(* PLC project product, Dassault Systèmes ControlBuild 2024x *)
(* stored: creationDateTime 2023-10-04T11:03:57-01:00 *)

(* This module simulates a generic product "box". *)
FUNCTION_BLOCK motion_control.product
  VAR
    status_act_prod : DINT := 0;
    m11 : REAL := 1.0;
    m12 : REAL := 0.0;
    m13 : REAL := 0.0;
    m14 : REAL := 0.0;
    m21 : REAL := 0.0;
    m22 : REAL := 1.0;
    m23 : REAL := 0.0;
    m24 : REAL := 0.0;
    m31 : REAL := 0.0;
    m32 : REAL := 0.0;
    m33 : REAL := 1.0;
    m34 : REAL := 0.0;
    m41 : REAL := 0.0;
    m42 : REAL := 0.0;
    m43 : REAL := 0.0;
    m44 : REAL := 1.0;
    movementConv : REAL := 0.0;
    contact : BOOL := false;
    centreRotX : REAL := 0.0;
    centreRotZ : REAL := 0.0;
    centreRotY : REAL := 0.0;
    moveDirection : INT := 0;
    idConv : DINT := 0;
    moveAuthorization : BOOL := false;
    number : INT := 0;
    idProdBelow : DINT := 0;
    prodId : INT := 0;
    oldOtherPx : REAL := 0.0;
    oldOtherPy : REAL := 0.0;
    oldOtherPz : REAL := 0.0;
    oldOtherRx : REAL := 0.0;
    oldOtherRy : REAL := 0.0;
    oldOtherRz : REAL := 0.0;
    gravitySpeed : REAL := 0.0;
    oldIdConv : DINT := 0;
  END_VAR
  VAR
    display1 : INT := 0;
    display2 : INT := 0;
    display3 : INT := 0;
    display4 : INT := 0;
    display5 : INT := 0;
    display6 : INT := 0;
    display7 : INT := 0;
    display8 : INT := 0;
    display9 : INT := 0;
    display10 : INT := 0;
  END_VAR
  VAR
    oPx : REAL := 0.0;
    oPy : REAL := 0.0;
    oPz : REAL := 0.0;
    oAx : REAL := 0.0;
    oAy : REAL := 0.0;
    oAz : REAL := 0.0;
    armActive : BOOL := false;
    memArmActive : BOOL := false;
    refAngZ : REAL := 0.0;
    refAngY : REAL := 0.0;
    refAngX : REAL := 0.0;
    refZ : REAL := 0.0;
    refY : REAL := 0.0;
    refX : REAL := 0.0;
    refSizeOthX : REAL := 0.0;
    refAngOthZ : REAL := 0.0;
    refAngOthY : REAL := 0.0;
    refAngOthX : REAL := 0.0;
    refOthZ : REAL := 0.0;
    refOthY : REAL := 0.0;
    refOthX : REAL := 0.0;
  END_VAR
  VAR
    empty1 : BOOL := false;
    empty2 : BOOL := false;
    empty3 : BOOL := false;
    empty4 : BOOL := false;
    empty5 : BOOL := false;
    empty6 : BOOL := false;
    empty7 : BOOL := false;
    empty8 : BOOL := false;
  END_VAR
  VAR
    weight : INT := 0;
  END_VAR


ACTION Prelude:
/* ----------------------------------------------------------------	*/
/* Initialisation of local variables of the instance of the product	*/
/* ----------------------------------------------------------------	*/
weight =0;
movementConv = 0.0;
contact = 0;
moveAuthorization = 1;
idConv=-1;
armActive = 0;

if (!empty1) weight +=15;
if (!empty2) weight +=15;
if (!empty3) weight +=15;
if (!empty4) weight +=15;
if (!empty5) weight +=15;
if (!empty6) weight +=15;
if (!empty7) weight +=15;
if (!empty8) weight +=15;
END_ACTION

ACTION Postlude:
/* ----------------------------------------------------------------	*/
/* If there is no contact, the box falls down thanks to gravity	*/	
/* ----------------------------------------------------------------	*/
if (contact == 0) 
	moveZBy(myself, gravitySpeed*-1.0);


/* ----------------------------------------------------------------	*/
/* Shift on conveyors if authorization					*/
/* ----------------------------------------------------------------	*/
if (moveAuthorization == 1 && (idConv>=0)) 
	moveRelativeAnotherBy(myself, idConv, movementConv, 0.0, 0.0);


/* ----------------------------------------------------------------	*/
/* Reset memories								*/
/* ----------------------------------------------------------------	*/
if (contact == 0) {
	moveDirection = 0;
	idProdBelow = -1;
}

memArmActive = armActive;
END_ACTION

ACTION motion_lib.qrreader:
otherVar(number) = number;
END_ACTION

ACTION motion_lib.weighingscale:
otherVar(weight) = weight;
END_ACTION

ACTION motion_lib.pusher:
moveBy(myself , otherVar(moveX1),otherVar(moveY1) , otherVar(moveZ1));
END_ACTION

ACTION motion_control.robotic_arm:
armActive = otherVar(functionActiveLocale);
if (armActive && !memArmActive ) {

// --- take arm/product relative position reference ---
	refOthX = getPositionX(other);
	refOthY = getPositionY(other);
	refOthZ = getPositionZ(other);
	refAngOthX = getAngleX(other);
	refAngOthY = getAngleY(other);
	refAngOthZ = getAngleZ(other);
	refSizeOthX = getSizeX(other);
	
	// move myself to the arm space reference 
	moveBy(myself, -refOthX, -refOthY, -refOthZ);

	rotateZBy(myself,-refAngOthZ,0.0, 0.0, 0.0);
	rotateYBy(myself,-refAngOthY,0.0, 0.0, 0.0);
	rotateXBy(myself,-refAngOthX,0.0, 0.0, 0.0);

	refX = getPositionX(myself);
	refY = getPositionY(myself);
	refZ = getPositionZ(myself);
	refAngX = getAngleX(myself);
	refAngY = getAngleY(myself);
	refAngZ = getAngleZ(myself);

	rotateBy(myself,refAngOthX,refAngOthY, refAngOthZ, 0.0, 0.0, 0.0); // relocate the product
	moveBy(myself, refOthX, refOthY, refOthZ);
}

if (armActive && memArmActive) {
	rotateTo(myself,refAngX,refAngY,refAngZ, getPositionX(myself), getPositionY(myself), getPositionZ(myself));
	moveTo(myself, refX, refY, refZ);
	rotateBy(myself,getAngleX(other),getAngleY(other), getAngleZ(other), 0.0, 0.0, 0.0);
	moveBy(myself, getPositionX(other), getPositionY(other), getPositionZ(other));

}
END_ACTION

ACTION motion_control.product_killer:
/* ----------------------------------------------------------------	*/
/* Destruction of the current instance of the product if the killer	*/
/* is active.									*/
/* ----------------------------------------------------------------	*/

if (otherVar(isActive)) prodKill(myself);
END_ACTION

ACTION motion_lib.conveyor:
/* ----------------------------------------------------------------	*/
/* Interaction between the product and conveyors			*/
/* Convention : a conveyor is always oriented so that its X-axis is	*/
/*	  	  in the same direction as the flow			*/
/* ----------------------------------------------------------------	*/

/* ----------------------------------------------------------------	*/
/* We retrieve the conveyor's data if the center of the product is	*/
/* included in the volume of the conveyor.				*/
/* ----------------------------------------------------------------	*/
if ((idConv == -1) || isMyCenterIncludedInXYOfOther(myself, other)) {
	/* Traverse speed on the conveyor	*/
	movementConv = otherVar(incShiftProduct) ;

	/* Keep trace of traverse direction of the conveyor		*/
	if (movementConv  > 0.0) moveDirection = DIR_FLOW;
	if (movementConv  < 0.0) moveDirection = DIR_INVERSE_FLOW;

	/* Get the identifier of the conveyor in order to be		*/
	/* able to shift the product in its coordinate system		*/
	idConv = other;
	oldIdConv = idConv;

	/* If the conveyor is a traverser, a lift, ...  		*/
	/* the product msut follow it	 				*/
	if (otherVar(incrementPositionX) != 0.0) moveXBy(myself, otherVar(incrementPositionX));
	if (otherVar(incrementPositionY) != 0.0) moveYBy(myself, otherVar(incrementPositionY));
	if (otherVar(incrementPositionZ) != 0.0) alignTwoObjectsRelativeThirdZ(myself, other, other);

	/* Management of the rotation of the product on a 		*/
	/* swivelling table, rotary plate ring, ...			*/
	/* Keep trace of the rotation center in order to be 		*/
	/* able to give them to products that could be stacked		*/
	/* above this instance						*/
	centreRotX = otherVar(centerRotX);
	centreRotY = otherVar(centerRotY);
	centreRotZ = otherVar(centerRotZ);

	if ((otherVar(incRotX) != 0.0) || (otherVar(incRotY)!= 0) || (otherVar(incRotZ)!= 0.0))
		rotateBy(myself, otherVar(incRotX), otherVar(incRotY), otherVar(incRotZ), centreRotX, centreRotY, centreRotZ);  

}

/* ----------------------------------------------------------------	*/
/* The product lays on a solid						*/
/* ----------------------------------------------------------------	*/
contact = 1;
END_ACTION

ACTION motion_lib.presence_sensor:
/* ----------------------------------------------------------------	*/
/* Information to the sensor that a product is in its detection area	*/
/* ----------------------------------------------------------------	*/

otherVar(detection) = 1;
END_ACTION

ACTION motion_control.product:
/* ----------------------------------------------------------------	*/
/* Interaction between two products	 				*/
/* ----------------------------------------------------------------	*/


/* Verify that the product whose position has to be updated is 	*/
/* located on one side of the current instance and not above or 	*/
/* below it.									*/
if ((getCenterZ(myself) > getCenterZ(other) - (getSizeZ(other)/2.0)) && (getCenterZ(myself) < getCenterZ(other)+(getSizeZ(other)/2.0))) {
	/* Update the position of the product that is behind the 	*/
	/* other according to the shift direction				*/
	if ( (moveDirection == DIR_FLOW && (getCenterXInAnother(myself, idConv) < getCenterXInAnother(other, idConv))) 
		|| (moveDirection == DIR_INVERSE_FLOW && (getCenterXInAnother(myself, idConv) > getCenterXInAnother(other, idConv))) ) {

		/* Align the 2 products one behind the other if its speed is lower 		*/
		if (fabs(movementConv ) > fabs(otherVar(movementConv )))
			alignTwoObjectsRelativeThirdX(myself, other, idConv);

		/* Forbid the shift						*/
		moveAuthorization=0;
	 }
}

/* Interaction with the product below					*/
if ((getCenterZ(myself)  > getCenterZ(other)+ (getSizeZ(other) / 2)) 
	&&  ((getCenterX(myself) > getCenterX(other) - (getSizeX(other)/4.0)) && (getCenterX(myself) < getCenterX(other)+(getSizeX(other)/4.0)))
	&&  ((getCenterY(myself) > getCenterY(other) - (getSizeY(other)/4.0)) && (getCenterY(myself) < getCenterY(other)+(getSizeY(other)/4.0))))  {
	/* Same movement than the product below				*/
	if (idProdBelow == other) {
		moveBy(myself, getPositionX(other)-oldOtherPx, getPositionY(other)-oldOtherPy, getPositionZ(other)-oldOtherPz);
		rotateBy(myself, getAngleX(other)-oldOtherRx, getAngleY(other)-oldOtherRy, getAngleZ(other)-oldOtherRz,
				otherVar(centreRotX), otherVar(centreRotY), otherVar(centreRotZ));
	}
	oldOtherPx=getPositionX(other); oldOtherPy=getPositionY(other); oldOtherPz=getPositionZ(other);
	oldOtherRx=getAngleX(other); oldOtherRy=getAngleY(other); oldOtherRz=getAngleZ(other);
	centreRotX=otherVar(centreRotX); centreRotY=otherVar(centreRotY); centreRotZ=otherVar(centreRotZ);

	idProdBelow = other;

	/* The product lays on a solid					*/
	contact = 1;

	/* The next line of code can be added in order to align 	*/
	/* correctly  the products one on the others ...		*/
	/* We should align both products in Z-axis according to the 	*/
	/* absolute coordinate system and not according to the 	*/
	/* relative system coordinate in order to have a generic 	*/
	/* behaviour.								*/
	/* => adapt this according to the application when needed	*/

	/* alignTwoObjectsRelativeThirdZ(myself, other, other); 	*/
	
}
END_ACTION

ACTION motion_control.product_creator:
/* ----------------------------------------------------------------	*/
/* Information to the creation module that a product is in its area	*/
/* ----------------------------------------------------------------	*/
 
otherVar(productPresence) = 1;
END_ACTION

ACTION C_header:
#define DIR_FLOW		1
#define DIR_INVERSE_FLOW	-1
END_ACTION
END_FUNCTION_BLOCK
